(* Generic TcpIp Connection  *) 
FUNCTION_BLOCK FB_TcpConnection
VAR_INPUT
	Ip					: T_IPv4Addr; (* IP Adress for TCP/IP Server *)
	Port 				: UDINT; (* Port To Connect to *)
	ReplyReadInterval 	: TIME := T#100MS; (* Time for allowing server to start responding [T#100MS]*)
END_VAR
VAR_OUTPUT
	_response 	: FB_StringBuilder;
END_VAR

VAR
	_requestAdr		: POINTER TO BYTE;
	_requestLength	: UDINT; 	
	
	_responseBuilder : FB_StringBuilder; 
	
	_responseString	: T_MAXSTRING; 
	_responseReceived	: BOOL; 
	_handle		: T_HSOCKET; 
	
	// ======== Current Connection
	_connect	: BOOL; 
	_connected	: BOOL; 

	_lastState		: E_TcpState; 
	_currentState	: E_TcpState :=  E_TcpState.Disconnected;

	// ======== ErrorString
	_errorID				: UDINT; 
	_errorMsg				: T_MAXSTRING; 

	// ======== Internal Stuff
	_idleTime	: TIME;
	_timeInState : TIME; 
	_stateCycles : UDINT;
	_firstTimeInState : BOOL; 
	
	// ======== Optional stuff
	_AmsNetId	: T_AmsNetID := ''; // Local host
	_Timeout	: TIME := T#45S; 
	
	
END_VAR

(*
Eventlog:
18-08-2018 - JHH - Created



*)


// ========== Initialize Buffers
_response.Initialize();

UpdateMetrics(	CurrentState 	:= _CurrentState,
				IdleTime		=> _IdleTime,
				TimeInState		=> _timeInState,
				CyclesInState 	=> _stateCycles, 
				FirstTimeInState => _firstTimeInState); 

_lastState := _currentState;
CASE _currentState OF
	// ============== Connect
		E_TcpState.Connecting:
			state_Connecting(		Handle			:= _handle,
									CurrentState	:= _currentState,
									Ip				:= Ip,
									Port			:= Port);	
		
		E_TcpState.Connected:
			state_Connected(		Connected		:= _connected); 
			
	// ============== Send/Receive	
		E_TcpState.Sending:

			state_Sending(			RequestAdr		:= _requestAdr,
									RequestLength	:= _requestLength,
									ResponseBuilder	:= _responseBuilder,
									CurrentState	:= _currentState,
									Handle			:= _handle);
									
								
									
		E_TcpState.Waiting:
			state_Waiting(			CurrentState	:= _currentState,
									WaitTime		:= ReplyReadInterval);
		
		E_TcpState.Receiving:

			state_Receiving(		ResponseBuilder := _responseBuilder,
									ActualResponse		:= _response,
									CurrentState	:= _currentState,
									Handle			:= _handle); 

						
		E_TcpState.Received:
			state_Received(			CurrentState	:= _currentState); 
									
	// ============== DisConnect							
		E_TcpState.Disconnecting:
			state_Disconnecting(	Handle			:= _handle,
									CurrentState	:= _currentState);	
	
		E_TcpState.Disconnected:
			state_Disconnected(		Connected		:= _connected);	
	
END_CASE

 
//_requestString := _request.ToString;


_errorMsg := ErrorIdToString(	ErrorID 		:= _errorID);

PROPERTY Busy : BOOL
GET
Busy := 	_currentState = E_TcpState.Receiving 
		OR	_currentState = E_TcpState.Sending
		OR	_currentState = E_TcpState.Waiting;
END_GET
END_PROPERTY

METHOD Connect : BOOL
IF _currentState = E_TcpState.Disconnected THEN
	_currentState := E_TcpState.Connecting; 
END_IF
END_METHOD

PROPERTY Connected : BOOL
GET
Connected := _connected;
END_GET
END_PROPERTY

METHOD Disconnect : BOOL
VAR_INPUT
END_VAR
_currentState := E_TcpState.Disconnecting;
END_METHOD

METHOD PRIVATE ErrorIdToString : T_MAXSTRING
VAR_INPUT
	ErrorID	: UDINT; 
END_VAR
CASE ErrorID OF
	0: 	
		ErrorIdToString := 'No Error';
	32769:
		ErrorIdToString := 'TCP/IP Connection Server: No new sockets can be created';
	32770:
		ErrorIdToString := 'TCP/IP Connection Server: Socket handle is invalid';
	32771:
		ErrorIdToString := 'TCP/IP Connection Server: TcpIp port listener already exists';
	32772:
		ErrorIdToString := 'TCP/IP Connection Server: Client socket is no longer connected with the server.';
	32773:
		ErrorIdToString := 'TCP/IP Connection Server: Error was registered in the listener socket.';
		
	2147952453:
		ErrorIdToString	:= 'Win32 Socket: An established connection was aborted BY the software in your host machine.';
		
	2147952454:
		ErrorIdToString	:= 'Win32 Socket: An existing connection was forcibly closed by the remote host..';
	 
ELSE
	ErrorIdToString := CONCAT('Unknown Error: ',TO_STRING(ErrorID));

END_CASE
END_METHOD

PROPERTY LastErrorMsg : T_MAXSTRING
GET
LastErrorMsg := _errorMsg;
END_GET
END_PROPERTY

METHOD PRIVATE MaintainConnection : BOOL
VAR_INPUT
	ServerIp		: T_IPv4Addr;
	ServerPort 		:  UDINT; 
	Connect			: BOOL; 
END_VAR

VAR_OUTPUT
	Handle				: T_HSOCKET; 
	ConnectionState		: E_SocketConnectionState; 
	Connected			: BOOL; 
	ErrorMsg			: T_MAXSTRING; 
END_VAR

VAR_INST
	_fbConnection		: FB_ClientServerConnection; 
	

END_VAR
_fbConnection(	sSrvNetID	:= , 
				nMode		:= 0, 
				sRemoteHost	:= ServerIp, 
				nRemotePort	:= ServerPort, 
				bEnable		:= Connect, 
				tReconnect	:= T#45S, 
				bBusy		=> , 
				bError		=> , 
				nErrId		=> , 
				hSocket		=> Handle, 
				eState		=> ConnectionState);
				
Connected := ConnectionState = 	E_SocketConnectionState.eSOCKET_CONNECTED;	
ErrorMsg := ErrorIdToString(_fbConnection.nErrId);
END_METHOD

METHOD ResetError : BOOL
_errorId := 0; 
_errorMsg := ErrorIdToString(_errorId);
END_METHOD

PROPERTY Response : REFERENCE TO FB_StringBuilder
GET
Response REF= _response;
END_GET
END_PROPERTY

PROPERTY ResponseReceived : BOOL
GET
ResponseReceived := _responseReceived;
END_GET
END_PROPERTY

METHOD Send : BOOL
VAR_INPUT
	RequestAdr	: POINTER TO BYTE;
	RequestLength	: UDINT; 
END_VAR
_responseBuilder.Clear();

_requestAdr	:= RequestAdr;
_requestLength := RequestLength; 

IF _currentState = E_TcpState.Connected THEN
	_currentState := E_TcpState.Sending;
END_IF
END_METHOD

PROPERTY State : E_TcpState
GET
State := _currentState;
END_GET
END_PROPERTY

METHOD private state_Connected : BOOL
VAR_IN_OUT
	Connected		: BOOL; 
END_VAR
Connected := TRUE;
END_METHOD

METHOD PRIVATE state_Connecting : BOOL
VAR_INPUT
	Ip					: T_IPv4Addr; (* IP Adress for TCP/IP Server *)
	Port 				: UDINT; (* Port To Connect to *)
END_VAR
VAR_IN_OUT
	Handle			: T_HSOCKET;
	CurrentState	: E_TcpState;		
END_VAR
VAR_INST
	fb				: FB_SocketConnect; 
	error			: T_MAXSTRING; 
END_VAR

fb(	sSrvNetId	:= _AmsNetId, 
	sRemoteHost	:= Ip, 
	nRemotePort	:= Port, 
	bExecute	:= NOT(_firstTimeInState), 
	tTimeout	:= _Timeout, 
	bBusy		=> , 
	bError		=> , 
	nErrId		=> , 
	hSocket		=> Handle);

IF fb.bError AND NOT(_firstTimeInState) THEN
	fb(bExecute := FALSE);
	error := ErrorIdToString(fb.nErrId); 
	CurrentState := E_TcpState.Disconnecting;

ELSIF NOT(fb.bBusy) AND NOT(_firstTimeInState) THEN
	fb(bExecute := FALSE);
	CurrentState := E_TcpState.Connected;
END_IF

_errorID := fb.nErrId;
END_METHOD

METHOD PRIVATE state_Disconnected : BOOL
VAR_IN_OUT
	Connected		: BOOL; 
END_VAR
Connected := FALSE; 
_connect := FALSE;
END_METHOD

METHOD private state_Disconnecting : BOOL
VAR_IN_OUT
	Handle			: T_HSOCKET;
	CurrentState	: E_TcpState;		
END_VAR
VAR_INST
	fb				: FB_SocketClose; 
	error 			: T_MAXSTRING;
END_VAR

fb(	sSrvNetId	:= _AmsNetId, 
	hSocket		:= Handle, 
	bExecute	:= NOT(_firstTimeInState), 
	tTimeout	:= _Timeout, 
	bBusy		=> , 
	bError		=> , 
	nErrId		=> );

IF (fb.bError OR NOT(fb.bBusy)) AND NOT(_firstTimeInState) THEN
	fb(bExecute := FALSE);
	error := ErrorIdToString(fb.nErrId); 
	CurrentState := E_TcpState.Disconnected;
END_IF

_errorID := fb.nErrId;
END_METHOD

METHOD state_Received : BOOL
VAR_IN_OUT
	CurrentState	: E_TcpState; 
END_VAR
IF NOT(_firstTimeInState) THEN
	CurrentState := E_TcpState.Connected; 
	
	_responseString 	:= _response.ToString; 
	_responseReceived	:= _response.Length > 0;

END_IF
END_METHOD

METHOD private state_Receiving : BOOL
VAR_IN_OUT
	ResponseBuilder	: FB_StringBuilder; 
	ActualResponse		: FB_StringBuilder;
END_VAR
VAR_IN_OUT
	Handle			: T_HSOCKET;
	CurrentState	: E_TcpState;		
END_VAR
VAR_INST
	fb				: FB_SocketReceive; 
	ErrorID			: UDINT; 
	TxtReceived		: T_MAXSTRING; 
	error 			: T_MAXSTRING;
	buffer			: ARRAY[0..1023] OF BYTE;
	InBuffer		: UDINT; 
END_VAR

fb(
	sSrvNetId	:= _AmsNetId, 
	hSocket		:= Handle, 
	bExecute	:= NOT(_firstTimeInState),
	cbLen		:= SIZEOF(buffer), //Response.BufferSize-Response.Length, 
	pDest		:= ADR(buffer), //Response.StringPointer + Response.Length, 
	tTimeout	:= T#500h, 
	bBusy		=> , 
	bError		=> , 
	nErrId		=> ErrorID, 
	nRecBytes	=> InBuffer); //BytesReceived);

IF fb.bError AND NOT(_firstTimeInState) THEN
	fb(bExecute := FALSE);
	error := ErrorIdToString(fb.nErrId); 
	CurrentState := E_TcpState.Disconnected;

ELSIF NOT(fb.bBusy) AND NOT(_firstTimeInState) THEN
	fb(bExecute := FALSE);
	
	// ========== Transfer to Response
	ResponseBuilder.AppendGeneric(ADR(buffer), InBuffer); 
	
	
	
	
	IF InBuffer > 0 THEN
		CurrentState := E_TcpState.Waiting;	// If not all bytes received, read again in "wait" time.
	ELSE
		CurrentState := E_TcpState.Received; // If no bytes read, reading is done. 
		TxtReceived := ResponseBuilder.ToString; 
		ActualResponse.Clear();
		ActualResponse.AppendGeneric(ResponseBuilder.StringPointer,ResponseBuilder.Length); 
	END_IF

END_IF

_errorID := fb.nErrId;
END_METHOD

METHOD PRIVATE state_Sending : BOOL
VAR_INPUT
	RequestAdr		: POINTER TO BYTE; 
	RequestLength	: UDINT; 
END_VAR
VAR_IN_OUT
	ResponseBuilder		: FB_StringBuilder;
	Handle			: T_HSOCKET;
	CurrentState	: E_TcpState;		
END_VAR

VAR_INST
	DebugRequest	: BOOL; 
	fb				: FB_SocketSend; 
	ErrorID			: UDINT; 
	RequestTxt		: T_MAXSTRING;
	error			: T_MAXSTRING;
END_VAR


fb(
		sSrvNetId	:= _AmsNetId, 
		hSocket		:= Handle, 
		bExecute	:= NOT(_firstTimeInState),
		cbLen		:= RequestLength, 
		pSrc		:= RequestAdr, 
		tTimeout	:= T#500h, 
		bBusy		=> , 
		bError		=> , 
		nErrId		=> ErrorID);
		


IF fb.bError AND NOT(_firstTimeInState) THEN
	fb(bExecute := FALSE);
	error := ErrorIdToString(fb.nErrId); 
	CurrentState := E_TcpState.Disconnected;

ELSIF NOT(fb.bBusy) AND NOT(_firstTimeInState) THEN
	fb(bExecute := FALSE);
	ResponseBuilder.Clear(); // Clear response, ready for receiving new response.
	CurrentState := E_TcpState.Waiting;
END_IF


_errorID := fb.nErrId;
END_METHOD

METHOD PRIVATE state_Waiting : BOOL
VAR_INPUT
	WaitTime	: TIME; 
END_VAR
VAR_IN_OUT
	CurrentState	: E_TcpState;
END_VAR
VAR_INST
	TimesExecuted : UDINT; 
END_VAR
IF WaitTime < T#5MS THEN
	WaitTime := T#50MS;
END_IF

IF _timeInState >= WaitTime THEN
	TimesExecuted := TimesExecuted + 1; 
	CurrentState := E_TcpState.Receiving; 
END_IF
END_METHOD

METHOD PRIVATE UpdateMetrics : BOOL
VAR_IN_OUT
	CurrentState	: E_TcpState; 	


END_VAR

VAR_OUTPUT
	IdleTime	: TIME; 	
	TimeInState	: TIME; 
	CyclesInState : UDINT;
	FirstTimeInState	 : BOOL; 
	
END_VAR

VAR_INST
	_lastState	: E_TcpState; 
	_IdleTimer	: TON; 
	_StateTimer	: TON; 
	_ReceiveTimer : TON;
	
	_cycles		: UDINT;
END_VAR

_IdleTimer(		IN	:= CurrentState = E_TcpState.Connected,
				PT	:= T#200H,
				ET	=> IdleTime); 

_StateTimer(	IN	:= CurrentState = _lastState,
				PT	:= T#1000H,
				ET	=> TimeInState); 
				
_ReceiveTimer(	IN	:= CurrentState = E_TcpState.Receiving OR CurrentState = E_TcpState.Waiting,
				PT	:= T#2S,	// Timeout for Receiving data
				ET	=> ); 
				
				
IF CurrentState = _lastState THEN
	_cycles := _cycles + 1;
	FirstTimeInState := FALSE;
ELSE
	_cycles := 0; 
	FirstTimeInState := TRUE; 
END_IF

IF _ReceiveTimer.Q OR _IdleTimer.ET > T#5s THEN
	CurrentState := E_TcpState.Disconnecting;
END_IF
				
CyclesInState := _cycles; 		
				
				
				
				
				
_lastState := CurrentState;
END_METHOD

END_FUNCTION_BLOCK

(* stored: Version 1.1.0.1, ProductVersion 3.1.4022.11
   POU FB_TcpConnection: Id {3d45db86-fe7a-4540-b3a7-dc04140d5100}, SpecialFunc None
   Folder Methods: Id {ea823e1a-d082-42dc-b7a3-2b16559d1185}
   Folder Properties: Id {5271c66d-3834-4504-af60-da9710c769c7}
   Folder states: Id {d32ea321-c335-46a2-b950-751aae19432d}
   Folder Utilities: Id {02681f13-a936-4722-9641-c3c90653d395}
   Property Busy: Id {cc2fb24b-f94b-4297-a5fe-e30ff41a5c71}
   Get Get: Id {84d73c8f-ba7d-42a5-b56e-83b5faae2dbc}
   Method Connect: Id {9db01490-a2dd-4726-91a3-be3a88e703a1}
   Property Connected: Id {2d3b838e-78d5-431c-b507-327f4d68e5e2}
   Get Get: Id {5579ad77-5229-4ae3-99c6-9bec769a8711}
   Method Disconnect: Id {97063573-256b-4ab0-adaa-68378975c270}
   Method ErrorIdToString: Id {10c2a147-9f20-4e79-adae-f9bb276e4728}
   Property LastErrorMsg: Id {33834a8e-462b-4b97-8e5c-342a557cef77}
   Get Get: Id {100f4272-bf66-40da-8b4a-854dbe706f65}
   Method MaintainConnection: Id {3bae8bd2-58fd-4151-926f-c10e1cb90010}
   Method ResetError: Id {7a928d15-19c3-42cb-8dbf-c5eaaf6c33ba}
   Property Response: Id {6195ca94-6009-4517-bc33-4a2aeab41dd4}
   Get Get: Id {7758283a-650c-4710-92ab-a821a5a930a9}
   Property ResponseReceived: Id {e24c3db4-37c7-4686-a745-14deae2b6137}
   Get Get: Id {155f97a7-fe52-4ce4-beef-51f6a13eba97}
   Method Send: Id {2cf89983-420b-473b-ab12-a784af3488b9}
   Property State: Id {91fc5d01-f365-4bd1-9760-d2758422b266}
   Get Get: Id {e838e9b8-8127-4fbb-b187-cce9e6633d33}
   Method state_Connected: Id {6fbfd44c-4f89-4c4e-b64f-0b24e16b90b8}
   Method state_Connecting: Id {acb82238-2349-4866-a293-6d86b2479460}
   Method state_Disconnected: Id {cf962620-1626-4b05-a4cc-8cd59d02909e}
   Method state_Disconnecting: Id {2d3c11da-96f8-4214-b966-d15009d033a1}
   Method state_Received: Id {48054237-e681-4146-bede-471942e910b0}
   Method state_Receiving: Id {e363cedc-2259-476b-a296-da630feeb833}
   Method state_Sending: Id {6124260b-37c8-4c96-a691-b0d64d14bc59}
   Method state_Waiting: Id {5b9f7827-0538-49b7-8f60-881a5290512a}
   Method UpdateMetrics: Id {8f62cb38-e43a-4e55-8455-e49872883a19} *)
